// TwinCAT 3 PLC project MC
// ProgramVersion: 3.1.4023.0
// libraries:
//   Tc2_MC2, * (Beckhoff Automation GmbH)
//   Tc2_Standard, * (Beckhoff Automation GmbH)
//   Tc2_System, * (Beckhoff Automation GmbH)
//   Tc3_Module, * (Beckhoff Automation GmbH)
//   VisuSymbols,3.5.10.0,System
// project tree:
//   / GlobalTextList.TcGTLO, PlcTask.TcTTO, 视图管理器.TcVMO (not stored)
//   POUs/ MAIN.TcPOU
// real-time tasks:
//   TASK PlcTask: cycle T#10ms, priority 20, ADS port 350
// motion (NC):
//   TASK NC-Task 1 SAF: cycle T#2ms, priority 4, ADS port 501
//   TASK NC-Task 1 SVB: cycle T#2ms, priority 8, ADS port 511
//   AXIS Axis 1 (id 1)
//     General: UnitName=°
//     Dynamic: AccelerationMaximum=3000, DecelerationMaximum=3000, Acceleration=40, Deceleration=40, Jerk=80
//     Velo: Fast=25, Maximum=25
//     OtherSettings: AllowMotionCmdToSlave=true
//     encoder EncType=19
//       EncPara: ScaleFactorNumerator=130321, ScaleFactorDenominator=40320000000, MaxCount=#xffffffff
//         SoftEndMinControl: Enable=true, Range=-96
//         SoftEndMaxControl: Enable=true, Range=96
//     drive DrvType=16
//       DrvPara: MaxCount=#xffffffff, DriveControlDWord=#x00020000
//         Analog: VeloReferenz=25, TorqueSetpointScale=10, ScaleFactorActTorque=0.1
//         TimeComp: TaskDelayCycles=1
//     controller CtrType=1
//       CtrPara: PriorControlFactor=1
//         Observer: BandWidth=20
// I/O:
//   DEVICE Device 3 (EtherCAT), AmsNetId 192.168.10.11.4.1
//     Box 1 (SSC-Device) [SSC-Device]
// variable links:
//   NC-Task 1 SAF/Axes/Axis 1 <-> Device 3 (EtherCAT)/Box 1 (SSC-Device)
//     Drive/Inputs/In/nState1 <-> ServoCntl Output TxPDO/Statusword
//     Drive/Inputs/In/nState2 <-> ServoCntl Output TxPDO/Statusword
//     Drive/Outputs/Out/nCtrl1 <-> ServoCntl Output RxPDO/Controlword
//     Drive/Outputs/Out/nDataOut1 <-> ServoCntl Output RxPDO/Target_position
//     Enc/Inputs/In/nDataIn1 <-> ServoCntl Output TxPDO/Position actual angle vaule
//   MC/MC Instance <-> NC-Task 1 SAF/Axes/Axis 1
//     PlcTask Inputs/MAIN.AXIS1.NcToPlc <-> Outputs/ToPlc
//     PlcTask Outputs/MAIN.AXIS1.PlcToNc <-> Inputs/FromPlc

CONFIGURATION MC
    RESOURCE PLC ON TwinCAT3
        TASK PlcTask(INTERVAL := T#10ms, PRIORITY := 20);
        PROGRAM MAIN WITH PlcTask : MAIN;
    END_RESOURCE
END_CONFIGURATION

// ---- POUs/MAIN.TcPOU
PROGRAM MAIN
VAR
	AXIS1:axis_ref;
	POWER1:mc_power;
	power_do: BOOL;

	move_abs: MC_MoveAbsolute;
	abs_do: BOOL;
	position: LREAL;
	vel: LREAL;
END_VAR

POWER1(
	Axis:= AXIS1, 
	Enable:= power_do, 
	Enable_Positive:= TRUE, 
	Enable_Negative:= TRUE, 
	Override:= , 
	BufferMode:= , 
	Options:= , 
	Status=> , 
	Busy=> , 
	Active=> , 
	Error=> , 
	ErrorID=> );
	
move_abs(
	Axis:= AXIS1, 
	Execute:= abs_do, 
	Position:= position, 
	Velocity:= vel, 
	Acceleration:= , 
	Deceleration:= , 
	Jerk:= , 
	BufferMode:= , 
	Options:= , 
	Done=> , 
	Busy=> , 
	Active=> , 
	CommandAborted=> , 
	Error=> , 
	ErrorID=> );

END_PROGRAM

// ---- GlobalTextList.TcGTLO
TEXTLIST GlobalTextList
  649 = '%f'
  315 = 'AXIS1:%.2F'
  472 = 'AXIS1:%.2f'
  845 = '使能'
  366 = '绝对运动'
END_TEXTLIST
